TYPE ST_BIT2 :
STRUCT
	a:BIT;
	b:BIT;
END_STRUCT
END_TYPE

(* stored: Version 1.1.0.1, ProductVersion 3.1.4024.12
   DUT ST_BIT2: Id {f07965de-c091-4aa2-b517-1cc77a3f3114} *)
